(* Logix 5000 project; controller R1USB70001_CWRU_Scenario_Gen_20111116 vendor 1 type 14 code 54 rev 19.11; software revision 19.01; part 6 of 9 *)
(* tags used below, declared in another part *)
   ExecutePv : ExecutePv;
   HMIPv : HMIPv;
   ControlMode : ControlModePub;
   EditScenario : EditScenarioPub;
   Execute : ExecutePub;
   HMI : HMIPub;
   HMI_Intfc_Read_Buffer : DINT[40];
   HMI_Intfc_String_Read_Buffer : STRING[2];
   HMI_Intfc_String_Write_Buffer : STRING;
   HMI_Intfc_Write_Buffer : DINT[20];
   Scenario : Scenario_Def[100];
(* MainProgram, continued *)

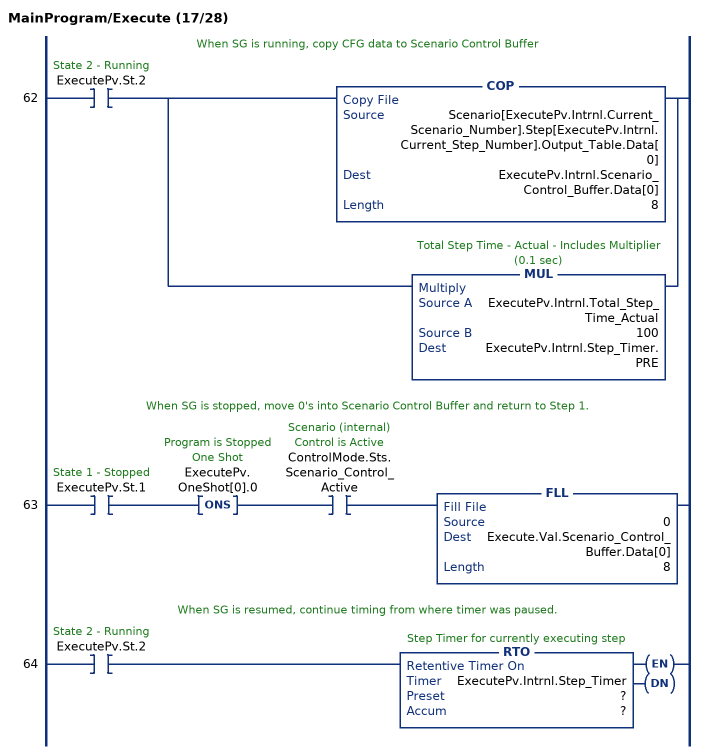
   // When SG is running, copy CFG data to Scenario Control Buffer
   62: XIC(ExecutePv.St.2)[COP(Scenario[ExecutePv.Intrnl.Current_Scenario_Number].Step[ExecutePv.Intrnl.Current_Step_Number].Output_Table.Data[0],ExecutePv.Intrnl.Scenario_Control_Buffer.Data[0],8) ,MUL(ExecutePv.Intrnl.Total_Step_Time_Actual,100,ExecutePv.Intrnl.Step_Timer.PRE) ];
   // When SG is stopped, move 0's into Scenario Control Buffer and return to Step 1.
   63: XIC(ExecutePv.St.1)ONS(ExecutePv.OneShot[0].0)XIC(ControlMode.Sts.Scenario_Control_Active)FLL(0,Execute.Val.Scenario_Control_Buffer.Data[0],8);
   // When SG is resumed, continue timing from where timer was paused.
   64: XIC(ExecutePv.St.2)RTO(ExecutePv.Intrnl.Step_Timer,?,?);
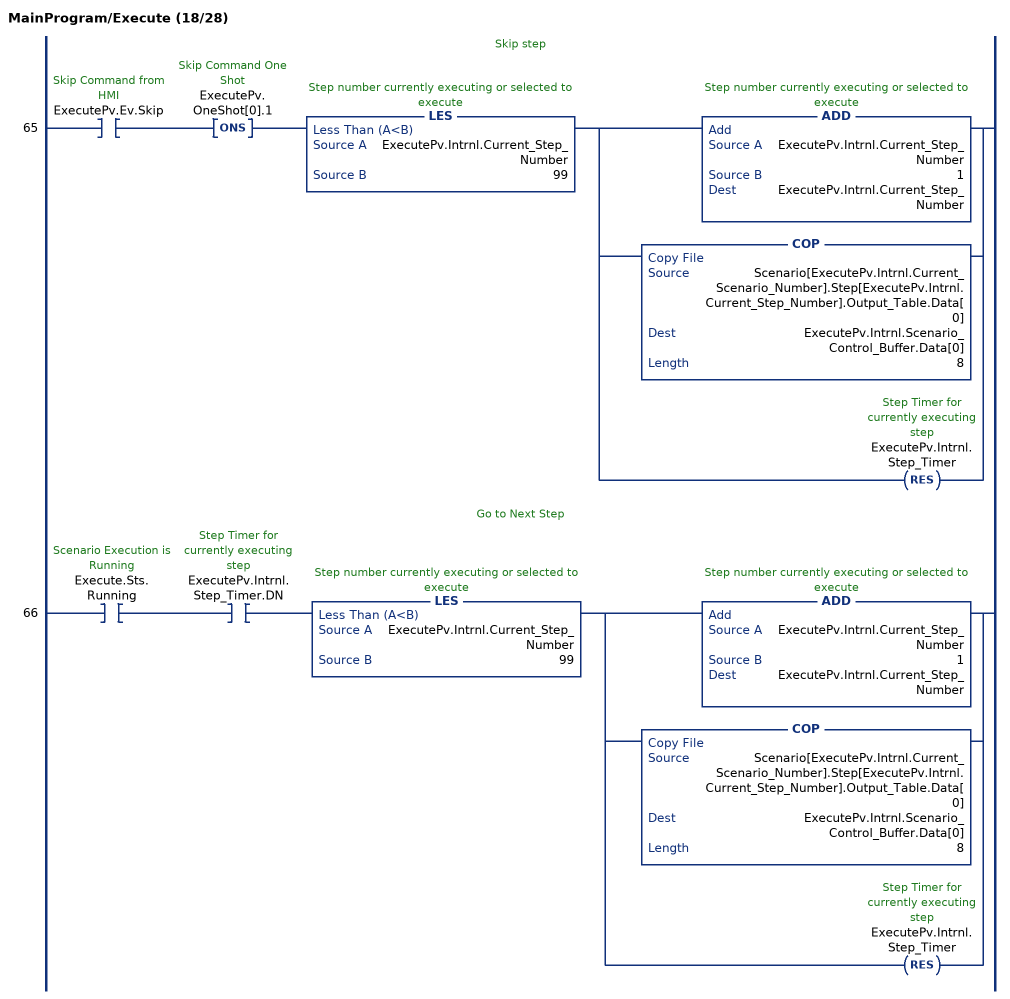
   // Skip step
   65: XIC(ExecutePv.Ev.Skip)ONS(ExecutePv.OneShot[0].1)LES(ExecutePv.Intrnl.Current_Step_Number,99)[ADD(ExecutePv.Intrnl.Current_Step_Number,1,ExecutePv.Intrnl.Current_Step_Number) ,COP(Scenario[ExecutePv.Intrnl.Current_Scenario_Number].Step[ExecutePv.Intrnl.Current_Step_Number].Output_Table.Data[0],ExecutePv.Intrnl.Scenario_Control_Buffer.Data[0],8) ,RES(ExecutePv.Intrnl.Step_Timer) ];
   // Go to Next Step
   66: XIC(Execute.Sts.Running)XIC(ExecutePv.Intrnl.Step_Timer.DN)LES(ExecutePv.Intrnl.Current_Step_Number,99)[ADD(ExecutePv.Intrnl.Current_Step_Number,1,ExecutePv.Intrnl.Current_Step_Number) ,COP(Scenario[ExecutePv.Intrnl.Current_Scenario_Number].Step[ExecutePv.Intrnl.Current_Step_Number].Output_Table.Data[0],ExecutePv.Intrnl.Scenario_Control_Buffer.Data[0],8) ,RES(ExecutePv.Intrnl.Step_Timer) ];
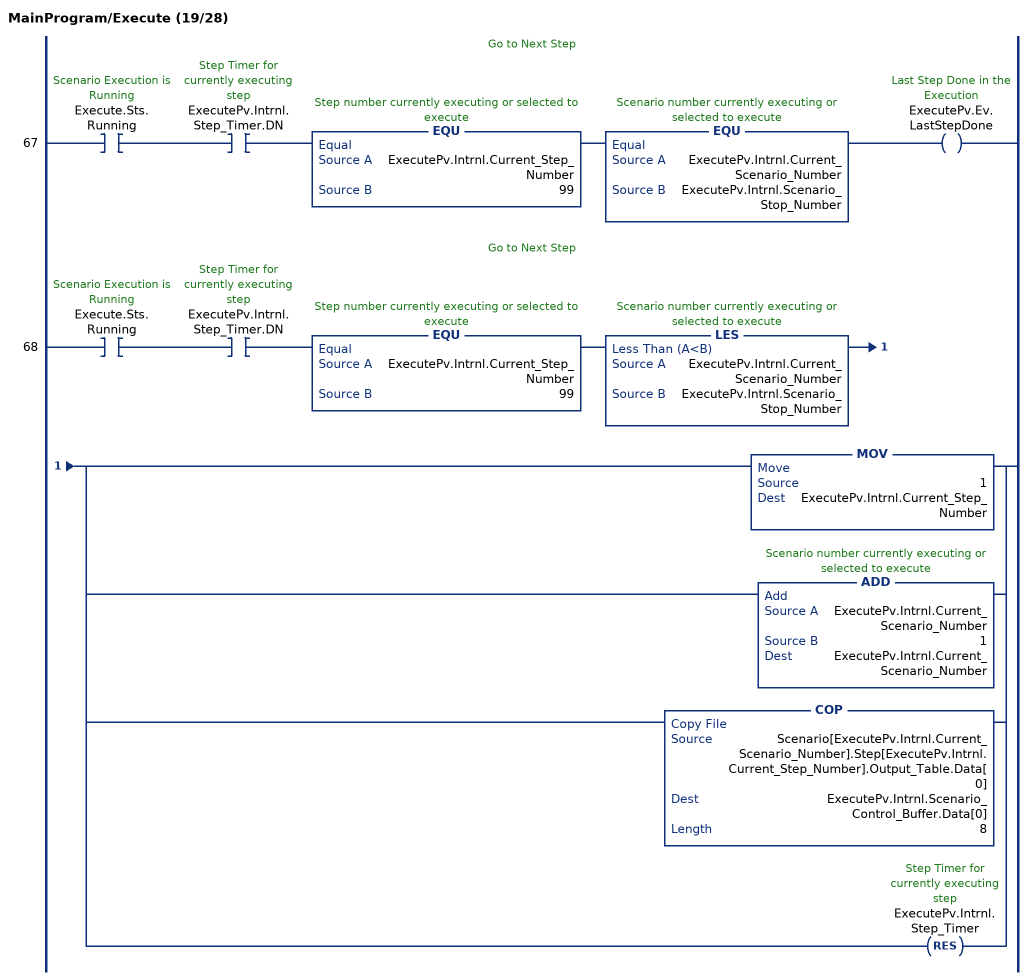
   // Go to Next Step
   67: XIC(Execute.Sts.Running)XIC(ExecutePv.Intrnl.Step_Timer.DN)EQU(ExecutePv.Intrnl.Current_Step_Number,99)EQU(ExecutePv.Intrnl.Current_Scenario_Number,ExecutePv.Intrnl.Scenario_Stop_Number)OTE(ExecutePv.Ev.LastStepDone);
   // Go to Next Step
   68: XIC(Execute.Sts.Running)XIC(ExecutePv.Intrnl.Step_Timer.DN)EQU(ExecutePv.Intrnl.Current_Step_Number,99)LES(ExecutePv.Intrnl.Current_Scenario_Number,ExecutePv.Intrnl.Scenario_Stop_Number)[MOV(1,ExecutePv.Intrnl.Current_Step_Number) ,ADD(ExecutePv.Intrnl.Current_Scenario_Number,1,ExecutePv.Intrnl.Current_Scenario_Number) ,COP(Scenario[ExecutePv.Intrnl.Current_Scenario_Number].Step[ExecutePv.Intrnl.Current_Step_Number].Output_Table.Data[0],ExecutePv.Intrnl.Scenario_Control_Buffer.Data[0],8) ,RES(ExecutePv.Intrnl.Step_Timer) ];
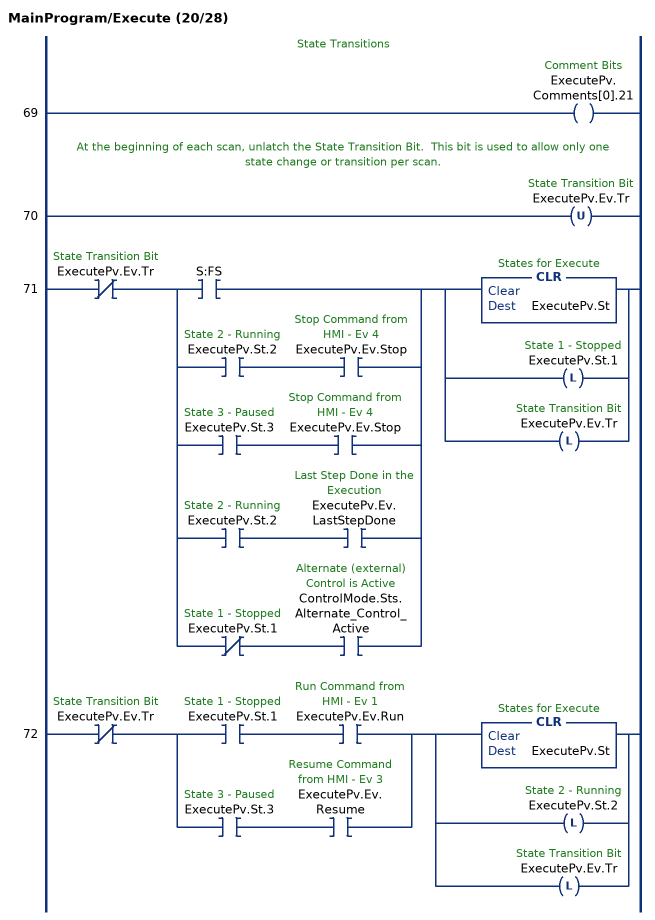
   // State Transitions
   69: OTE(ExecutePv.Comments[0].21);
   // At the beginning of each scan, unlatch the State Transition Bit.  This bit is used to allow only one state change or transition per scan.
   70: OTU(ExecutePv.Ev.Tr);
   71: XIO(ExecutePv.Ev.Tr)[XIC(S:FS) ,XIC(ExecutePv.St.2) XIC(ExecutePv.Ev.Stop) ,XIC(ExecutePv.St.3) XIC(ExecutePv.Ev.Stop) ,XIC(ExecutePv.St.2) XIC(ExecutePv.Ev.LastStepDone) ,XIO(ExecutePv.St.1) XIC(ControlMode.Sts.Alternate_Control_Active) ][CLR(ExecutePv.St) ,OTL(ExecutePv.St.1) ,OTL(ExecutePv.Ev.Tr) ];
   72: XIO(ExecutePv.Ev.Tr)[XIC(ExecutePv.St.1) XIC(ExecutePv.Ev.Run) ,XIC(ExecutePv.St.3) XIC(ExecutePv.Ev.Resume) ][CLR(ExecutePv.St) ,OTL(ExecutePv.St.2) ,OTL(ExecutePv.Ev.Tr) ];
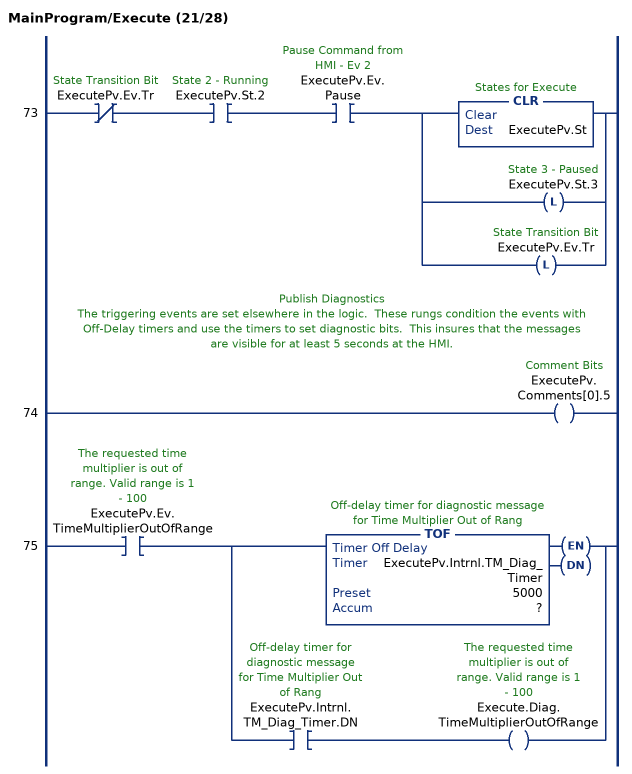
   73: XIO(ExecutePv.Ev.Tr)XIC(ExecutePv.St.2)XIC(ExecutePv.Ev.Pause)[CLR(ExecutePv.St) ,OTL(ExecutePv.St.3) ,OTL(ExecutePv.Ev.Tr) ];
   // Publish Diagnostics
   // The triggering events are set elsewhere in the logic.  These rungs condition the events with Off-Delay timers and use the timers to set diagnostic bits.  This insures that the messages are visible for at least 5 seconds at the HMI.
   74: OTE(ExecutePv.Comments[0].5);
   75: XIC(ExecutePv.Ev.TimeMultiplierOutOfRange)[TOF(ExecutePv.Intrnl.TM_Diag_Timer,?,?) ,XIC(ExecutePv.Intrnl.TM_Diag_Timer.DN) OTE(Execute.Diag.TimeMultiplierOutOfRange) ];
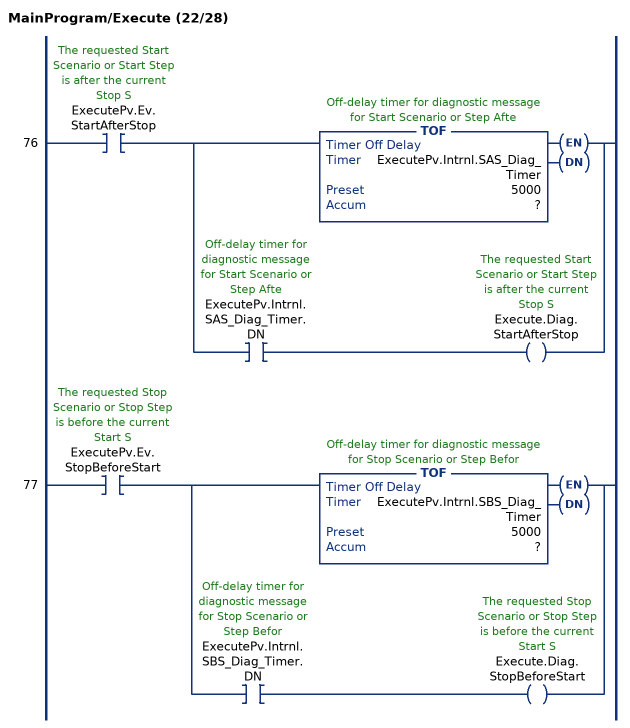
   76: XIC(ExecutePv.Ev.StartAfterStop)[TOF(ExecutePv.Intrnl.SAS_Diag_Timer,?,?) ,XIC(ExecutePv.Intrnl.SAS_Diag_Timer.DN) OTE(Execute.Diag.StartAfterStop) ];
   77: XIC(ExecutePv.Ev.StopBeforeStart)[TOF(ExecutePv.Intrnl.SBS_Diag_Timer,?,?) ,XIC(ExecutePv.Intrnl.SBS_Diag_Timer.DN) OTE(Execute.Diag.StopBeforeStart) ];
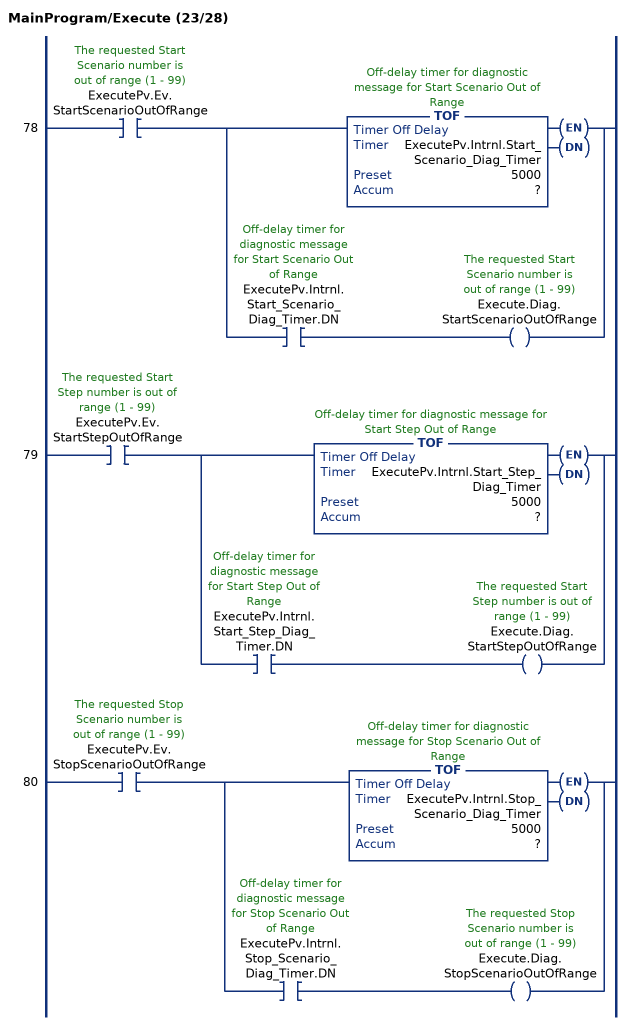
   78: XIC(ExecutePv.Ev.StartScenarioOutOfRange)[TOF(ExecutePv.Intrnl.Start_Scenario_Diag_Timer,?,?) ,XIC(ExecutePv.Intrnl.Start_Scenario_Diag_Timer.DN) OTE(Execute.Diag.StartScenarioOutOfRange) ];
   79: XIC(ExecutePv.Ev.StartStepOutOfRange)[TOF(ExecutePv.Intrnl.Start_Step_Diag_Timer,?,?) ,XIC(ExecutePv.Intrnl.Start_Step_Diag_Timer.DN) OTE(Execute.Diag.StartStepOutOfRange) ];
   80: XIC(ExecutePv.Ev.StopScenarioOutOfRange)[TOF(ExecutePv.Intrnl.Stop_Scenario_Diag_Timer,?,?) ,XIC(ExecutePv.Intrnl.Stop_Scenario_Diag_Timer.DN) OTE(Execute.Diag.StopScenarioOutOfRange) ];
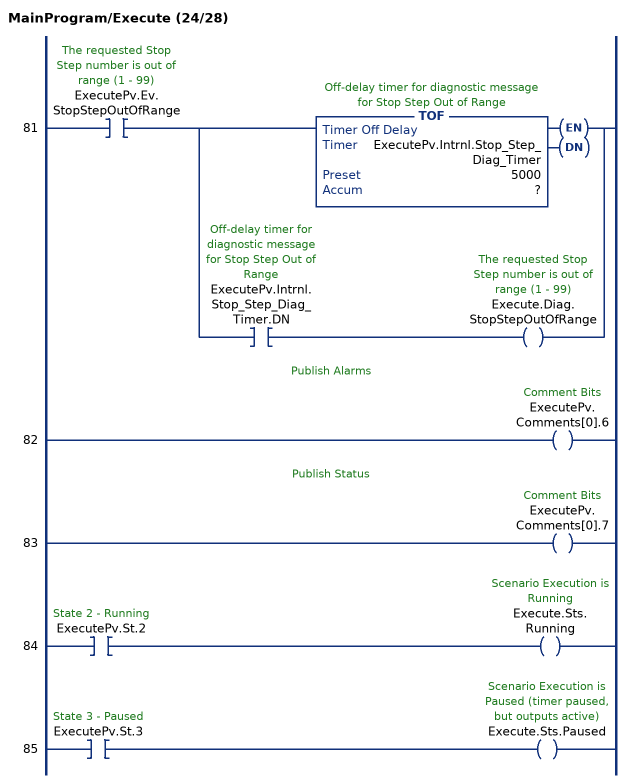
   81: XIC(ExecutePv.Ev.StopStepOutOfRange)[TOF(ExecutePv.Intrnl.Stop_Step_Diag_Timer,?,?) ,XIC(ExecutePv.Intrnl.Stop_Step_Diag_Timer.DN) OTE(Execute.Diag.StopStepOutOfRange) ];
   // Publish Alarms
   82: OTE(ExecutePv.Comments[0].6);
   // Publish Status
   83: OTE(ExecutePv.Comments[0].7);
   84: XIC(ExecutePv.St.2)OTE(Execute.Sts.Running);
   85: XIC(ExecutePv.St.3)OTE(Execute.Sts.Paused);
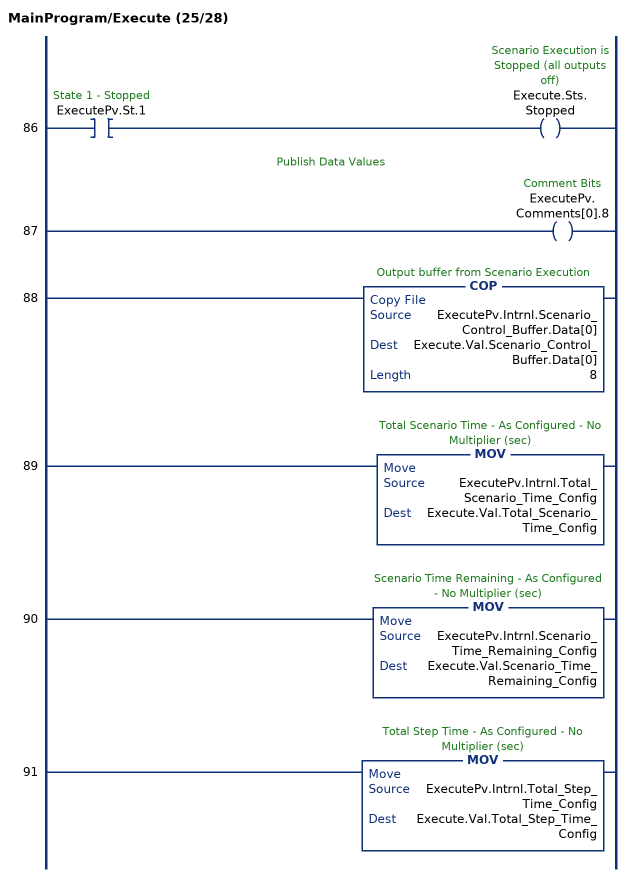
   86: XIC(ExecutePv.St.1)OTE(Execute.Sts.Stopped);
   // Publish Data Values
   87: OTE(ExecutePv.Comments[0].8);
   88: COP(ExecutePv.Intrnl.Scenario_Control_Buffer.Data[0],Execute.Val.Scenario_Control_Buffer.Data[0],8);
   89: MOV(ExecutePv.Intrnl.Total_Scenario_Time_Config,Execute.Val.Total_Scenario_Time_Config);
   90: MOV(ExecutePv.Intrnl.Scenario_Time_Remaining_Config,Execute.Val.Scenario_Time_Remaining_Config);
   91: MOV(ExecutePv.Intrnl.Total_Step_Time_Config,Execute.Val.Total_Step_Time_Config);
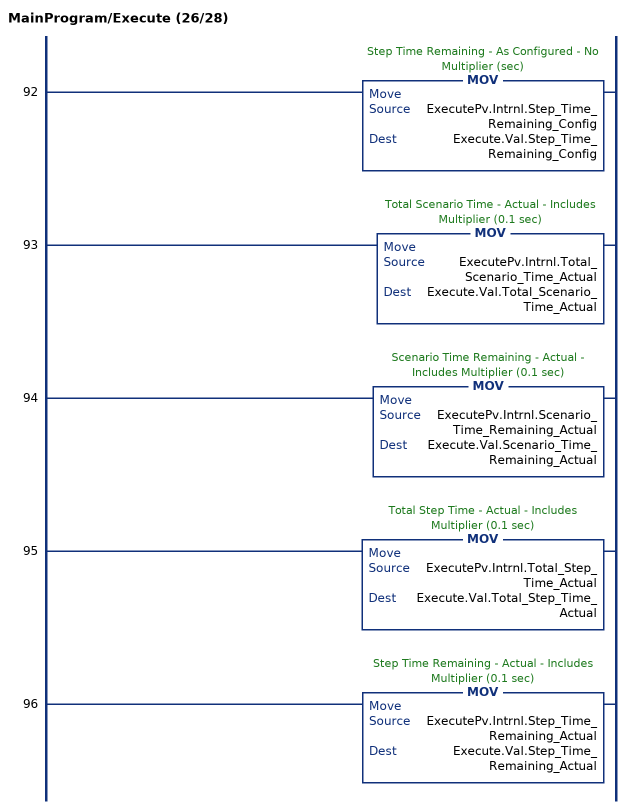
   92: MOV(ExecutePv.Intrnl.Step_Time_Remaining_Config,Execute.Val.Step_Time_Remaining_Config);
   93: MOV(ExecutePv.Intrnl.Total_Scenario_Time_Actual,Execute.Val.Total_Scenario_Time_Actual);
   94: MOV(ExecutePv.Intrnl.Scenario_Time_Remaining_Actual,Execute.Val.Scenario_Time_Remaining_Actual);
   95: MOV(ExecutePv.Intrnl.Total_Step_Time_Actual,Execute.Val.Total_Step_Time_Actual);
   96: MOV(ExecutePv.Intrnl.Step_Time_Remaining_Actual,Execute.Val.Step_Time_Remaining_Actual);
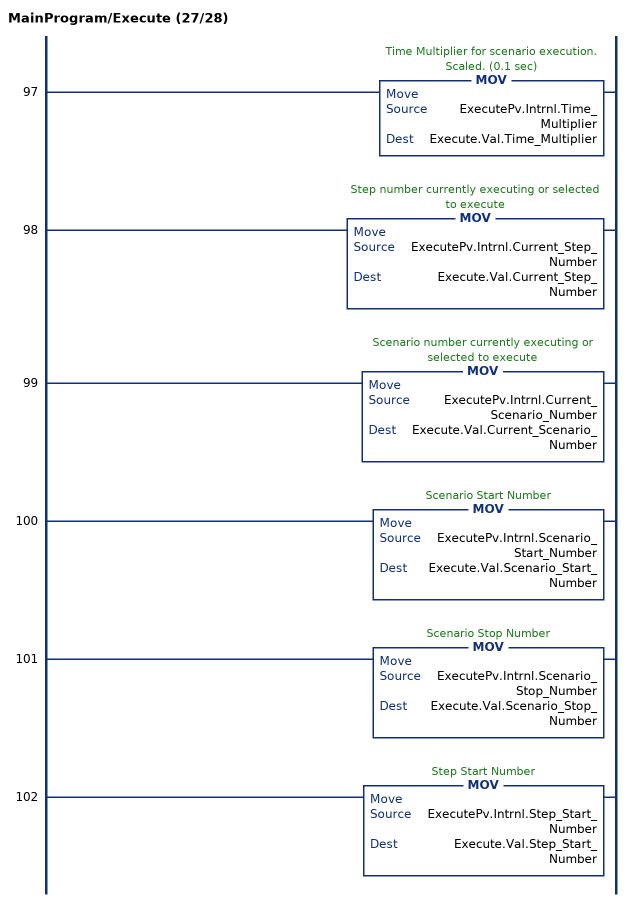
   97: MOV(ExecutePv.Intrnl.Time_Multiplier,Execute.Val.Time_Multiplier);
   98: MOV(ExecutePv.Intrnl.Current_Step_Number,Execute.Val.Current_Step_Number);
   99: MOV(ExecutePv.Intrnl.Current_Scenario_Number,Execute.Val.Current_Scenario_Number);
   100: MOV(ExecutePv.Intrnl.Scenario_Start_Number,Execute.Val.Scenario_Start_Number);
   101: MOV(ExecutePv.Intrnl.Scenario_Stop_Number,Execute.Val.Scenario_Stop_Number);
   102: MOV(ExecutePv.Intrnl.Step_Start_Number,Execute.Val.Step_Start_Number);
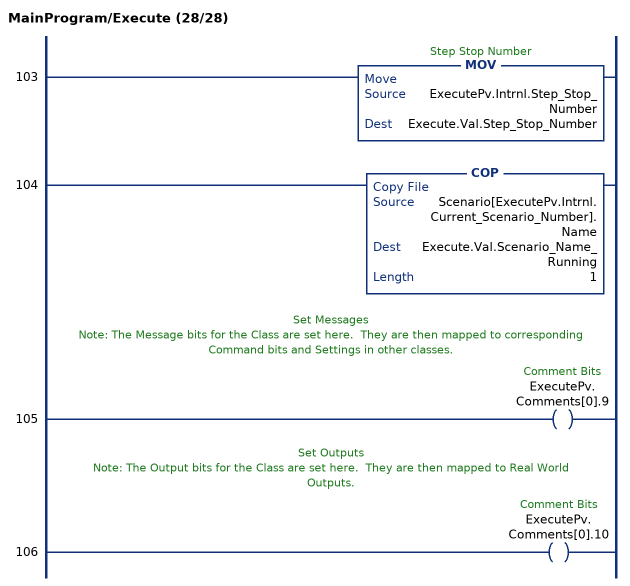
   103: MOV(ExecutePv.Intrnl.Step_Stop_Number,Execute.Val.Step_Stop_Number);
   104: COP(Scenario[ExecutePv.Intrnl.Current_Scenario_Number].Name,Execute.Val.Scenario_Name_Running,1);
   // Set Messages
   // Note: The Message bits for the Class are set here.  They are then mapped to corresponding Command bits and Settings in other classes.
   105: OTE(ExecutePv.Comments[0].9);
   // Set Outputs
   // Note: The Output bits for the Class are set here.  They are then mapped to Real World Outputs.
   106: OTE(ExecutePv.Comments[0].10);
END_ROUTINE

ROUTINE HMI   (* ladder *)
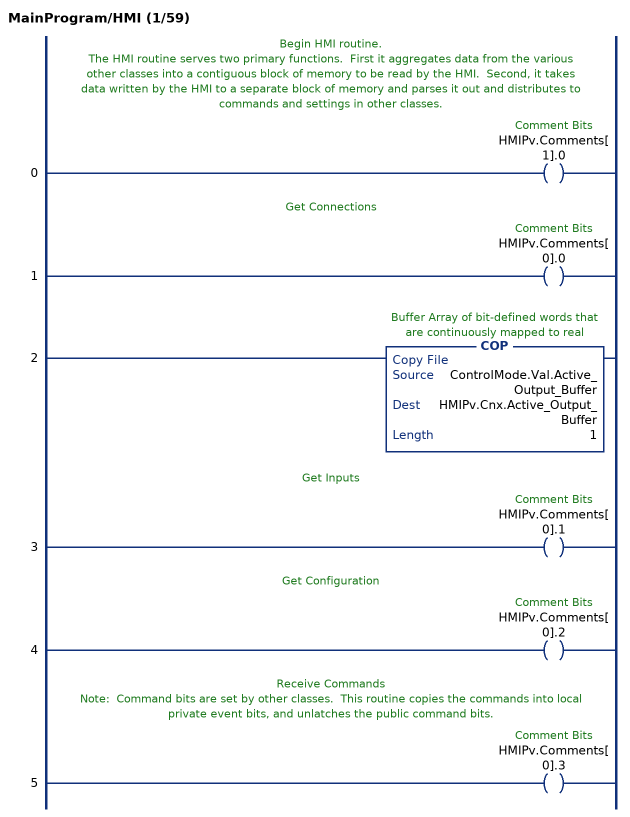
   // Begin HMI routine.
   // The HMI routine serves two primary functions.  First it aggregates data from the various other classes into a contiguous block of memory to be read by the HMI.  Second, it takes data written by the HMI to a separate block of memory and parses it out and distributes to commands and settings in other classes.
   0: OTE(HMIPv.Comments[1].0);
   // Get Connections
   1: OTE(HMIPv.Comments[0].0);
   2: COP(ControlMode.Val.Active_Output_Buffer,HMIPv.Cnx.Active_Output_Buffer,1);
   // Get Inputs
   3: OTE(HMIPv.Comments[0].1);
   // Get Configuration
   4: OTE(HMIPv.Comments[0].2);
   // Receive Commands
   // Note:  Command bits are set by other classes.  This routine copies the commands into local private event bits, and unlatches the public command bits.
   5: OTE(HMIPv.Comments[0].3);
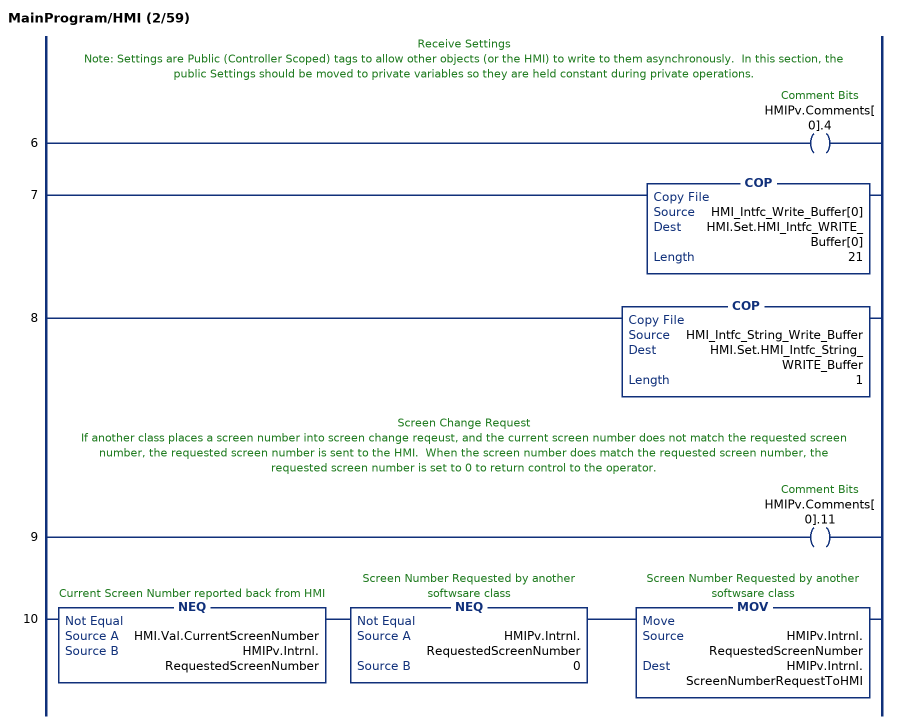
   // Receive Settings
   // Note: Settings are Public (Controller Scoped) tags to allow other objects (or the HMI) to write to them asynchronously.  In this section, the public Settings should be moved to private variables so they are held constant during private operations.
   6: OTE(HMIPv.Comments[0].4);
   7: COP(HMI_Intfc_Write_Buffer[0],HMI.Set.HMI_Intfc_WRITE_Buffer[0],21);
   8: COP(HMI_Intfc_String_Write_Buffer,HMI.Set.HMI_Intfc_String_WRITE_Buffer,1);
   // Screen Change Request
   // If another class places a screen number into screen change reqeust, and the current screen number does not match the requested screen number, the requested screen number is sent to the HMI.  When the screen number does match the requested screen number, the requested screen number is set to 0 to return control to the operator.
   9: OTE(HMIPv.Comments[0].11);
   10: NEQ(HMI.Val.CurrentScreenNumber,HMIPv.Intrnl.RequestedScreenNumber)NEQ(HMIPv.Intrnl.RequestedScreenNumber,0)MOV(HMIPv.Intrnl.RequestedScreenNumber,HMIPv.Intrnl.ScreenNumberRequestToHMI);
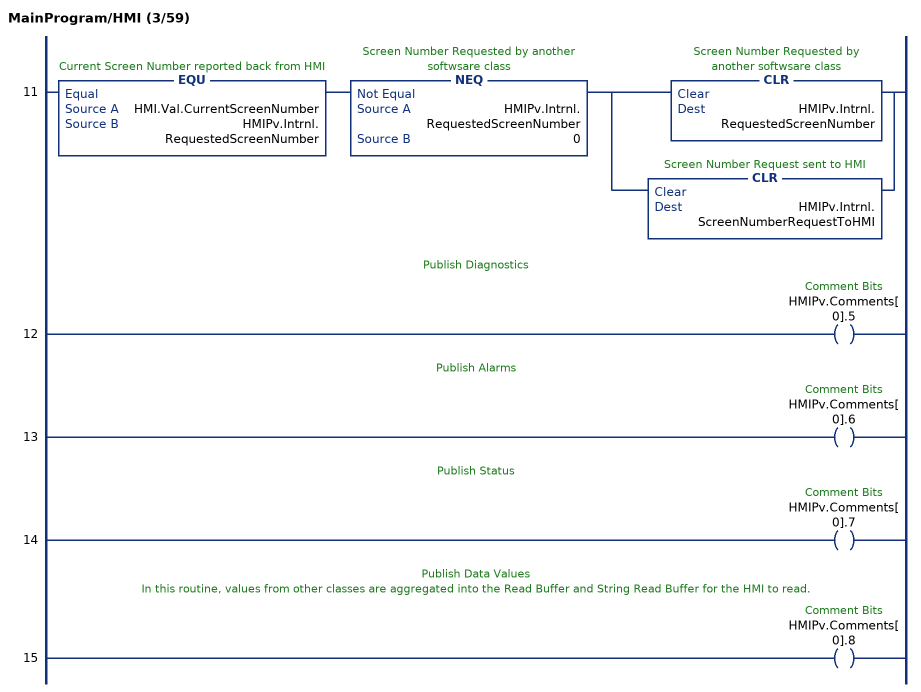
   11: EQU(HMI.Val.CurrentScreenNumber,HMIPv.Intrnl.RequestedScreenNumber)NEQ(HMIPv.Intrnl.RequestedScreenNumber,0)[CLR(HMIPv.Intrnl.RequestedScreenNumber) ,CLR(HMIPv.Intrnl.ScreenNumberRequestToHMI) ];
   // Publish Diagnostics
   12: OTE(HMIPv.Comments[0].5);
   // Publish Alarms
   13: OTE(HMIPv.Comments[0].6);
   // Publish Status
   14: OTE(HMIPv.Comments[0].7);
   // Publish Data Values
   // In this routine, values from other classes are aggregated into the Read Buffer and String Read Buffer for the HMI to read.
   15: OTE(HMIPv.Comments[0].8);
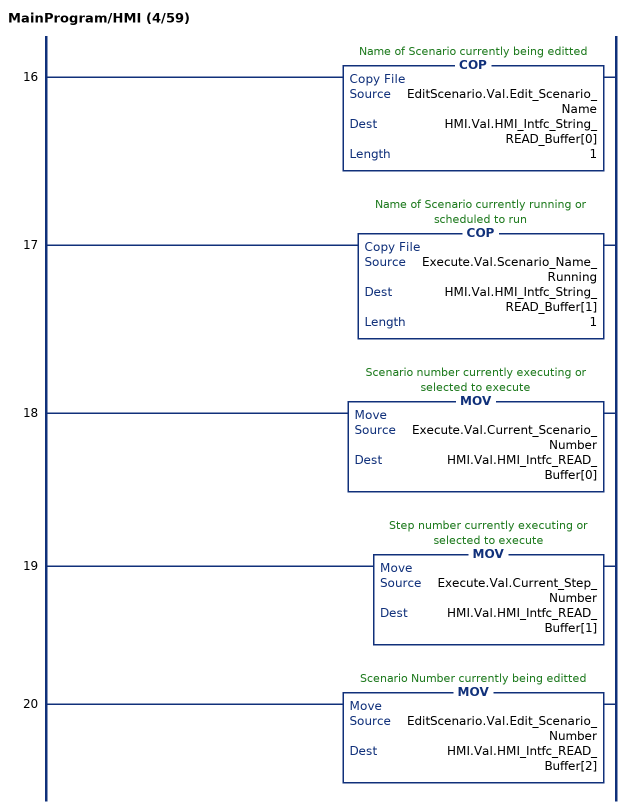
   16: COP(EditScenario.Val.Edit_Scenario_Name,HMI.Val.HMI_Intfc_String_READ_Buffer[0],1);
   17: COP(Execute.Val.Scenario_Name_Running,HMI.Val.HMI_Intfc_String_READ_Buffer[1],1);
   18: MOV(Execute.Val.Current_Scenario_Number,HMI.Val.HMI_Intfc_READ_Buffer[0]);
   19: MOV(Execute.Val.Current_Step_Number,HMI.Val.HMI_Intfc_READ_Buffer[1]);
   20: MOV(EditScenario.Val.Edit_Scenario_Number,HMI.Val.HMI_Intfc_READ_Buffer[2]);
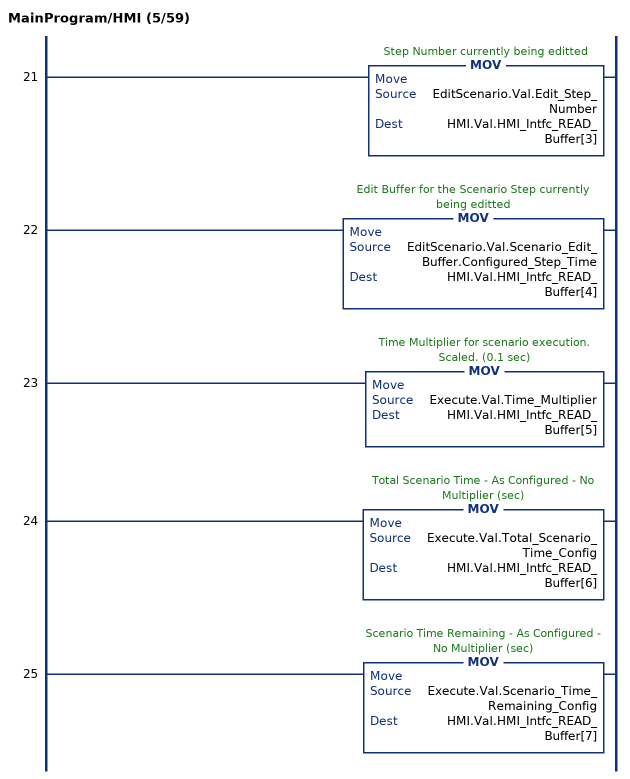
   21: MOV(EditScenario.Val.Edit_Step_Number,HMI.Val.HMI_Intfc_READ_Buffer[3]);
   22: MOV(EditScenario.Val.Scenario_Edit_Buffer.Configured_Step_Time,HMI.Val.HMI_Intfc_READ_Buffer[4]);
   23: MOV(Execute.Val.Time_Multiplier,HMI.Val.HMI_Intfc_READ_Buffer[5]);
   24: MOV(Execute.Val.Total_Scenario_Time_Config,HMI.Val.HMI_Intfc_READ_Buffer[6]);
   25: MOV(Execute.Val.Scenario_Time_Remaining_Config,HMI.Val.HMI_Intfc_READ_Buffer[7]);
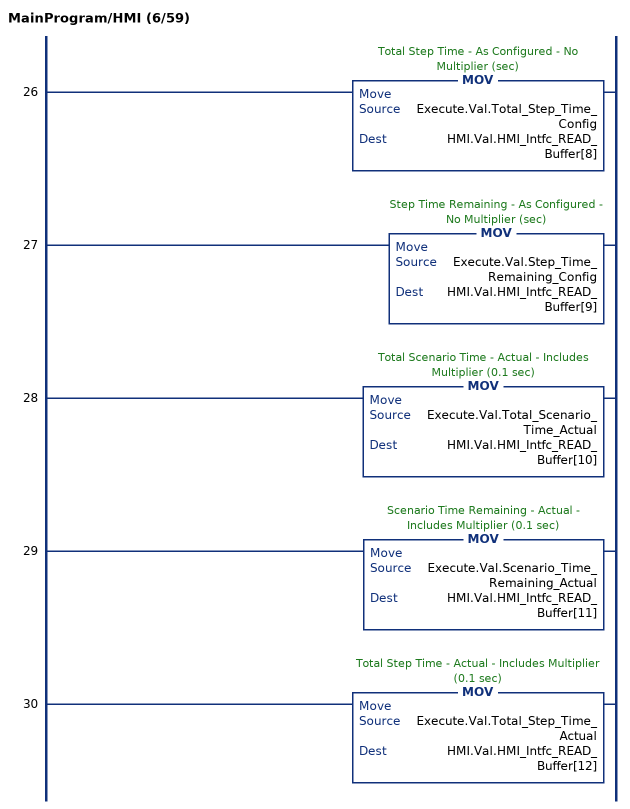
   26: MOV(Execute.Val.Total_Step_Time_Config,HMI.Val.HMI_Intfc_READ_Buffer[8]);
   27: MOV(Execute.Val.Step_Time_Remaining_Config,HMI.Val.HMI_Intfc_READ_Buffer[9]);
   28: MOV(Execute.Val.Total_Scenario_Time_Actual,HMI.Val.HMI_Intfc_READ_Buffer[10]);
   29: MOV(Execute.Val.Scenario_Time_Remaining_Actual,HMI.Val.HMI_Intfc_READ_Buffer[11]);
   30: MOV(Execute.Val.Total_Step_Time_Actual,HMI.Val.HMI_Intfc_READ_Buffer[12]);
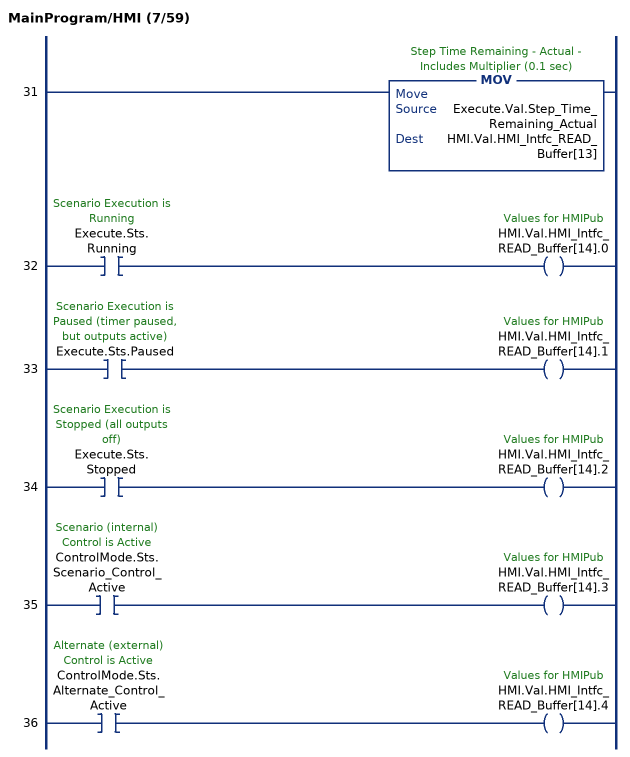
   31: MOV(Execute.Val.Step_Time_Remaining_Actual,HMI.Val.HMI_Intfc_READ_Buffer[13]);
   32: XIC(Execute.Sts.Running)OTE(HMI.Val.HMI_Intfc_READ_Buffer[14].0);
   33: XIC(Execute.Sts.Paused)OTE(HMI.Val.HMI_Intfc_READ_Buffer[14].1);
   34: XIC(Execute.Sts.Stopped)OTE(HMI.Val.HMI_Intfc_READ_Buffer[14].2);
   35: XIC(ControlMode.Sts.Scenario_Control_Active)OTE(HMI.Val.HMI_Intfc_READ_Buffer[14].3);
   36: XIC(ControlMode.Sts.Alternate_Control_Active)OTE(HMI.Val.HMI_Intfc_READ_Buffer[14].4);
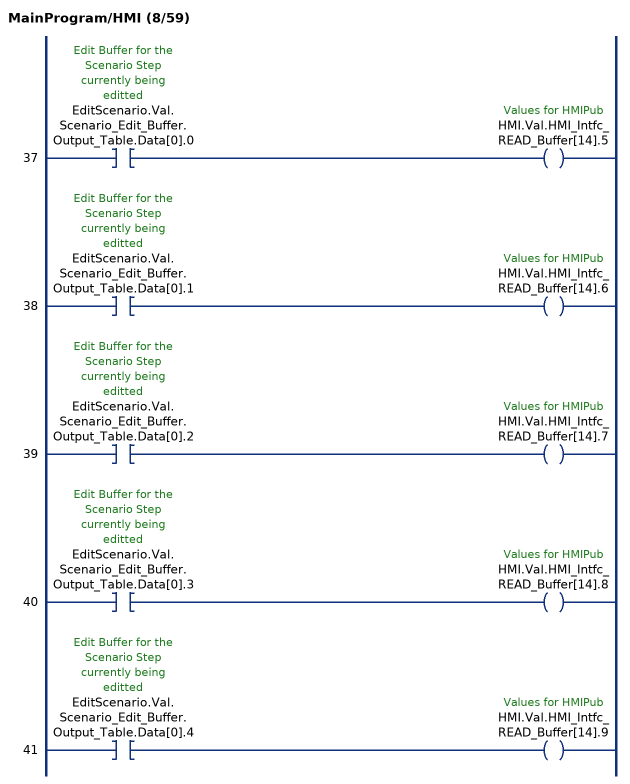
   37: XIC(EditScenario.Val.Scenario_Edit_Buffer.Output_Table.Data[0].0)OTE(HMI.Val.HMI_Intfc_READ_Buffer[14].5);
   38: XIC(EditScenario.Val.Scenario_Edit_Buffer.Output_Table.Data[0].1)OTE(HMI.Val.HMI_Intfc_READ_Buffer[14].6);
   39: XIC(EditScenario.Val.Scenario_Edit_Buffer.Output_Table.Data[0].2)OTE(HMI.Val.HMI_Intfc_READ_Buffer[14].7);
   40: XIC(EditScenario.Val.Scenario_Edit_Buffer.Output_Table.Data[0].3)OTE(HMI.Val.HMI_Intfc_READ_Buffer[14].8);
   41: XIC(EditScenario.Val.Scenario_Edit_Buffer.Output_Table.Data[0].4)OTE(HMI.Val.HMI_Intfc_READ_Buffer[14].9);
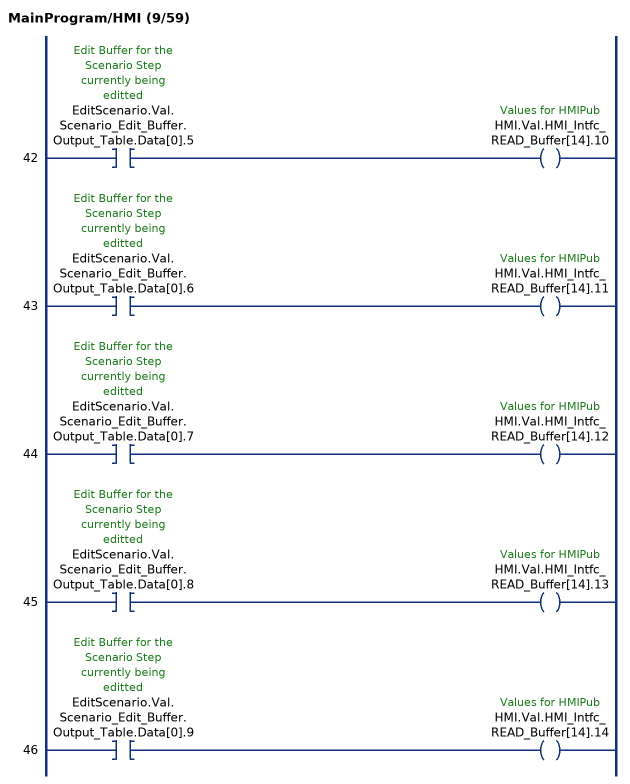
   42: XIC(EditScenario.Val.Scenario_Edit_Buffer.Output_Table.Data[0].5)OTE(HMI.Val.HMI_Intfc_READ_Buffer[14].10);
   43: XIC(EditScenario.Val.Scenario_Edit_Buffer.Output_Table.Data[0].6)OTE(HMI.Val.HMI_Intfc_READ_Buffer[14].11);
   44: XIC(EditScenario.Val.Scenario_Edit_Buffer.Output_Table.Data[0].7)OTE(HMI.Val.HMI_Intfc_READ_Buffer[14].12);
   45: XIC(EditScenario.Val.Scenario_Edit_Buffer.Output_Table.Data[0].8)OTE(HMI.Val.HMI_Intfc_READ_Buffer[14].13);
   46: XIC(EditScenario.Val.Scenario_Edit_Buffer.Output_Table.Data[0].9)OTE(HMI.Val.HMI_Intfc_READ_Buffer[14].14);
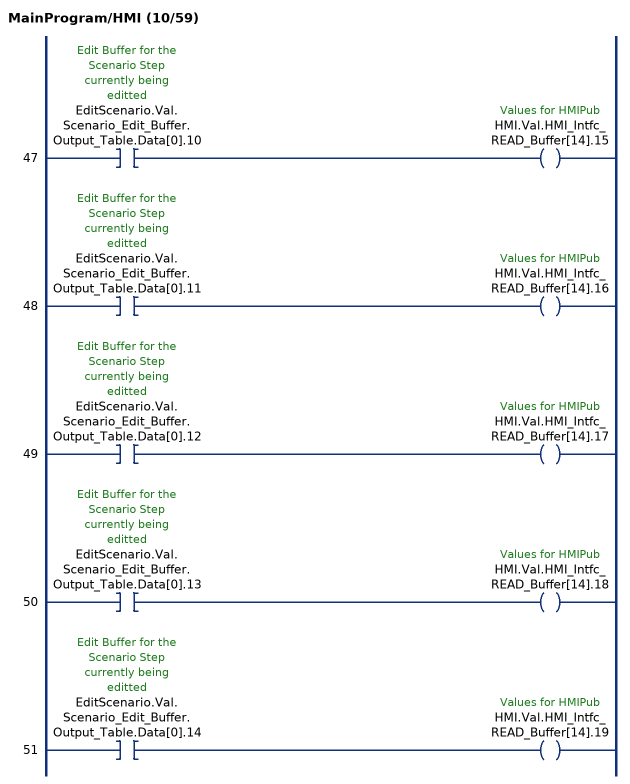
   47: XIC(EditScenario.Val.Scenario_Edit_Buffer.Output_Table.Data[0].10)OTE(HMI.Val.HMI_Intfc_READ_Buffer[14].15);
   48: XIC(EditScenario.Val.Scenario_Edit_Buffer.Output_Table.Data[0].11)OTE(HMI.Val.HMI_Intfc_READ_Buffer[14].16);
   49: XIC(EditScenario.Val.Scenario_Edit_Buffer.Output_Table.Data[0].12)OTE(HMI.Val.HMI_Intfc_READ_Buffer[14].17);
   50: XIC(EditScenario.Val.Scenario_Edit_Buffer.Output_Table.Data[0].13)OTE(HMI.Val.HMI_Intfc_READ_Buffer[14].18);
   51: XIC(EditScenario.Val.Scenario_Edit_Buffer.Output_Table.Data[0].14)OTE(HMI.Val.HMI_Intfc_READ_Buffer[14].19);
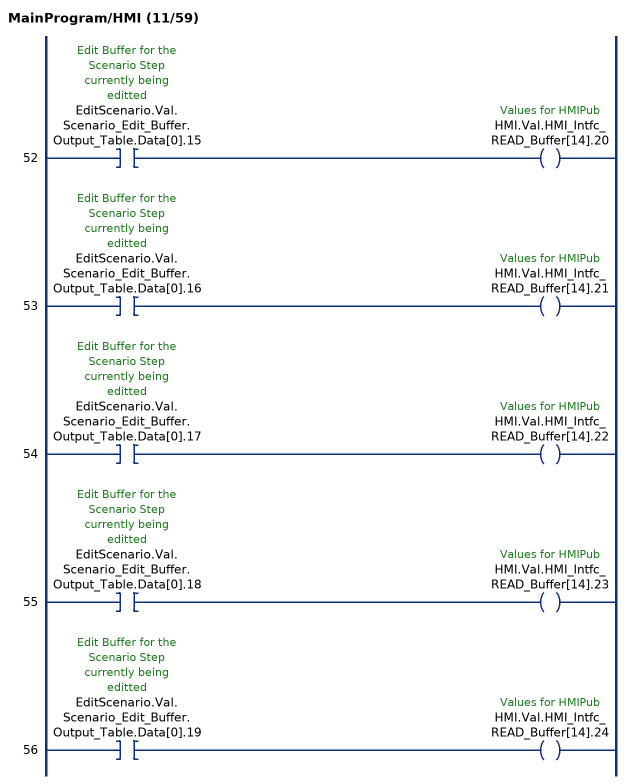
   52: XIC(EditScenario.Val.Scenario_Edit_Buffer.Output_Table.Data[0].15)OTE(HMI.Val.HMI_Intfc_READ_Buffer[14].20);
   53: XIC(EditScenario.Val.Scenario_Edit_Buffer.Output_Table.Data[0].16)OTE(HMI.Val.HMI_Intfc_READ_Buffer[14].21);
   54: XIC(EditScenario.Val.Scenario_Edit_Buffer.Output_Table.Data[0].17)OTE(HMI.Val.HMI_Intfc_READ_Buffer[14].22);
   55: XIC(EditScenario.Val.Scenario_Edit_Buffer.Output_Table.Data[0].18)OTE(HMI.Val.HMI_Intfc_READ_Buffer[14].23);
   56: XIC(EditScenario.Val.Scenario_Edit_Buffer.Output_Table.Data[0].19)OTE(HMI.Val.HMI_Intfc_READ_Buffer[14].24);
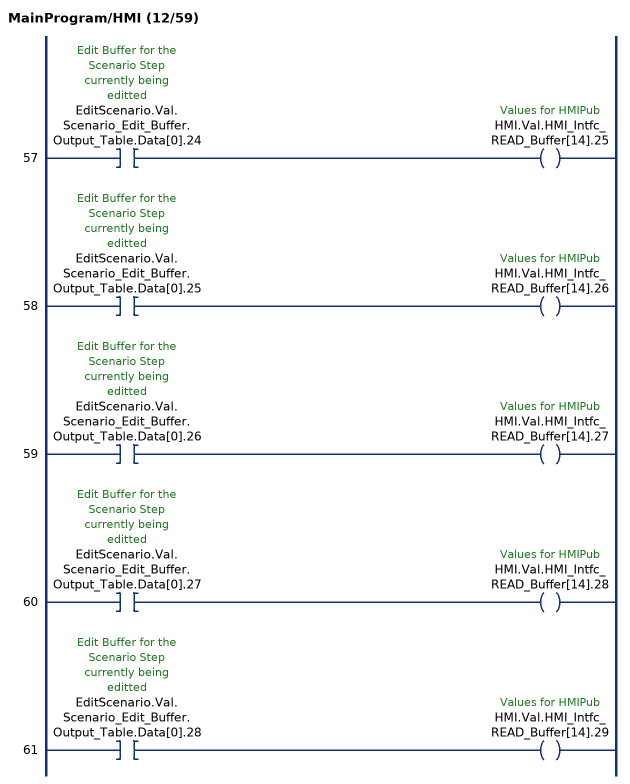
   57: XIC(EditScenario.Val.Scenario_Edit_Buffer.Output_Table.Data[0].24)OTE(HMI.Val.HMI_Intfc_READ_Buffer[14].25);
   58: XIC(EditScenario.Val.Scenario_Edit_Buffer.Output_Table.Data[0].25)OTE(HMI.Val.HMI_Intfc_READ_Buffer[14].26);
   59: XIC(EditScenario.Val.Scenario_Edit_Buffer.Output_Table.Data[0].26)OTE(HMI.Val.HMI_Intfc_READ_Buffer[14].27);
   60: XIC(EditScenario.Val.Scenario_Edit_Buffer.Output_Table.Data[0].27)OTE(HMI.Val.HMI_Intfc_READ_Buffer[14].28);
   61: XIC(EditScenario.Val.Scenario_Edit_Buffer.Output_Table.Data[0].28)OTE(HMI.Val.HMI_Intfc_READ_Buffer[14].29);
